(* CoDeSys 2.3 export: TYPE_INPUTS.EXP *)

(* Data type *)
TYPE TYPE_INPUTS :
	STRUCT
		TasteAusfahren: BOOL;
		TasteEinfahren: BOOL;
		TastePoweredByGenerator: BOOL;
		EndschalterNotantrieb: BOOL;
		EndschalterEingefahren: BOOL;
		EndschalterAufgerichtet: BOOL;
	END_STRUCT
END_TYPE
